// TIA Portal V19 export
TYPE "C501_STU_PMP_TYPIC"
   STRUCT
      CMD { ExternalAccessible := 'False'; ExternalVisible := 'False'; ExternalWritable := 'False'} : USInt;   // Sturing pomp
      LCK_AAN { ExternalAccessible := 'False'; ExternalVisible := 'False'; ExternalWritable := 'False'} : Bool;   // TRUE = Vergrendelen pomp (ook in manueel en hand)
      CMD_SNE { ExternalAccessible := 'False'; ExternalVisible := 'False'; ExternalWritable := 'False'} : Real;   // Sturing snelheid pomp
   END_STRUCT;
END_TYPE
